RoboDK station: Übung2.rdk

Station Übung2 (saved by RoboDK 5.6.9). Poses are relative to the parent item; angles as X-Y-Z fixed-axis rotations.
  - frame world at (0, 0, 0) mm
    - frame F1 at (0, 1000, 0) mm, rotated rx 0 ry -90 rz 90 deg
      - frame F2 at (0, 1000, 0) mm, rotated rx 90 ry 0 rz 90 deg
    - frame check at (-1000, 1000, 0) mm, rotated rx 0 ry 0 rz 180 deg
  - Python program Prog1 (listed below)

--- Python program Prog1 ---
# Type help("robodk.robolink") or help("robodk.robomath") for more information
# Press F5 to run the script
# Documentation: https://robodk.com/doc/en/RoboDK-API.html
# Reference:     https://robodk.com/doc/en/PythonAPI/robodk.html
# Note: It is not required to keep a copy of this file, your Python script is saved with your RDK project
from robodk.robolink import *      # RoboDK API
from robodk.robomath import *    # Robot link toolbox

# Link to RoboDK
RDK = Robolink()

robot = RDK.Item('Staubli TX2-40')

world = RDK.Item('world')
home = RDK.Item('home')
target1 = RDK.Item('Target 1')
target2 = RDK.Item('Target 2')
target3 = RDK.Item('Target 3')

print('start')

robot.setAccelerationJoints(150)
robot.setSpeedJoints(150)

#
robot.setSpeed(50, 50, 150, 150)

robot.MoveJ(home)
robot.MoveJ(target1) # PTP T1
robot.MoveL(target2) # LIN T2
robot.MoveC(target1, target3) # CIR T3 via T1
robot.MoveL(target2) # LIN T2
robot.MoveJ(target1) # PTP T1
robot.MoveJ(home) # PTP home

print('end')
